// TIA Portal V20 export
FUNCTION_BLOCK "FB_PrioSequence"   // FB79, SCL
{ S7_Optimized_Access := 'TRUE' }
// stored: MemoryReserve 100, SetENOAutomatically false
   VAR
      sPrio : Int;
   END_VAR
BEGIN
   REGION Description header 
       //==================================================================================
       // POSALUX Swiss SA / (C) Copyright 2026
       //----------------------------------------------------------------------------------
       // Title: 
       // Comment/Function: FB_PrioSequence
       // Author: Fabien WALDT
       // Engineering: TIA Portal v20
       //----------------------------------------------------------------------------------
       // Change log table:
       // Version  | Date     | Expert in charge | Changes applied
       // ---------|----------|------------------|-----------------------------------------
       // 00.00.01 | 20260205 | WFA              | First released version
       // =================================================================================
   END_REGION

   REGION Test Prio
       // #sPrio := 0;

       // IF "DB_LoaderShuttle1".sMain.sInterface.SequenceRun AND "DB_LoaderShuttle2".sMain.sInterface.SequenceRun THEN
       //     IF "DB_LoaderShuttle2".sMain.sCurrent_Step_NB > "DB_LoaderShuttle1".sMain.sCurrent_Step_NB THEN
       //         #sPrio := 2;
       //     ELSE
       //         #sPrio := 1;
       //     END_IF;
       // ELSIF "DB_LoaderShuttle1".sMain.sInterface.SequenceRun AND NOT "DB_LoaderShuttle2".sMain.sInterface.SequenceRun THEN
       //     #sPrio := 1;
       // ELSIF NOT "DB_LoaderShuttle1".sMain.sInterface.SequenceRun AND "DB_LoaderShuttle2".sMain.sInterface.SequenceRun THEN
       //     #sPrio := 2;
       // ELSE
       //     #sPrio := 0;
       // END_IF;
       // 
       IF "DB_HMISetting".Shuttle1Enable AND NOT "DB_HMISetting".Shuttle2Enable THEN
           #sPrio := 1;
       ELSIF "DB_HMISetting".Shuttle2Enable AND NOT "DB_HMISetting".Shuttle1Enable THEN
           #sPrio := 2;
       ELSIF "DB_HMISetting".Shuttle1Enable AND NOT "DB_HMISetting".Shuttle2Enable AND "DB_LoaderShuttle2".sMain.sCurrent_Step_NB > "DB_LoaderShuttle1".sMain.sCurrent_Step_NB THEN
           #sPrio := 2;
       ELSE
           #sPrio := 1;
       END_IF;
   END_REGION
END_FUNCTION_BLOCK
